FUNCTION_BLOCK T_AdsRead
VAR
    _Execution : T_Execution;
    AdsRead1 : ADSREAD := (TMOUT := T#2S);
END_VAR

IF _Execution.Aborting THEN
    _Execution.SetAborted();
END_IF

AdsRead1(
	NETID:= , 
	PORT:= , 
	IDXGRP:= , 
	IDXOFFS:= , 
	LEN:= , 
	DESTADDR:= , 
	READ:= _Execution.Starting, 
	TMOUT:= , 
	BUSY=> , 
	ERR=> , 
	ERRID=> );

    
IF _Execution.Starting THEN
    _Execution.SetBusy();
END_IF
IF _Execution.Busy AND NOT AdsRead1.BUSY THEN
    IF AdsRead1.ERR THEN
        _Execution.SetError(AdsRead1.ERRID);
    ELSE
        _Execution.SetDone();
	END_IF
END_IF

METHOD Execute : BOOL
VAR_INPUT
	AmsNetId:T_AmsNetid;
	Port:T_AmsPort;
	IndexGroup:UDINT; 
	IndexOffset:UDINT;
	DataLength:UDINT; 
	DataAddress:PVOID; 
END_VAR
AdsRead1.NETID      := AmsNetId;
AdsRead1.PORT       := Port;
AdsRead1.IDXGRP     := IndexGroup;
AdsRead1.IDXOFFS    := IndexOffset;
AdsRead1.LEN        := DataLength;
AdsRead1.DESTADDR   := DataAddress;

Execute := _Execution.Start();
END_METHOD

PROPERTY Execution : I_Execution
GET
Execution := _Execution;
END_GET
END_PROPERTY

END_FUNCTION_BLOCK

(* stored: Version 1.1.0.1, ProductVersion 3.1.4024.6
   POU T_AdsRead: Id {58f6bcea-8104-4956-ae95-3413ce461b25}, SpecialFunc None
   Method Execute: Id {27ab2939-d629-482d-b359-f86144e5ccf1}
   Property Execution: Id {2c86a2d0-0e71-4e17-b0f8-f799e350876d}
   Get Get: Id {babe62a8-694f-4fc4-8cb0-2753944348e5} *)
